Omron CX-Programmer project NuevoProyecto (CX-Programmer 9.61)

# PLC Caramelos: CJ2M CPU11

## Program NuevoPrograma1 (cyclic task 0)
Local symbols
CincoCent 1.01 BOOL  ; 1.01
DiezCent 1.02 BOOL  ; 1.02
Encender 0.00 BOOL  ; 0.00
ExpulsandoCaA 1.14 BOOL  ; 1.14
ExpulsandoCaB 1.15 BOOL  ; 1.15
IgualQueCinco 3.11 BOOL  ; 3.11
IgualQueDiez 3.12 BOOL  ; 3.12
IgualQueQuince 3.03 BOOL  ; 3.03
IgualQueVeinte 3.02 BOOL  ; 3.02
LedCarameloA 1.06 BOOL  ; 1.06
LedCarameloB 1.07 BOOL  ; 1.07
MasDeVeinte 1.05 BOOL  ; 1.05
MayorQueVeinte 3.10 BOOL  ; 3.10
MenorQueVeinte 3.01 BOOL  ; 3.01
P0 2.00 BOOL  ; 2.00
P1 2.01 BOOL  ; 2.01
P2 2.02 BOOL  ; 2.02
P3 2.03 BOOL  ; 2.03
P4 2.04 BOOL  ; 2.04
P5 2.05 BOOL  ; 2.05
P6 2.06 BOOL  ; 2.06
P7 2.07 BOOL  ; 2.07
P8 2.08 BOOL  ; 2.08
P9 2.09 BOOL  ; 2.09
Preparada 1.00 BOOL  ; 1.00
QuinceCent 1.03 BOOL  ; 1.03
Recuperar 0.11 BOOL  ; 0.11
Reset 2.10 BOOL  ; 2.10
SeleccionarCaA 0.14 BOOL  ; 0.14
SeleccionarCaB 0.15 BOOL  ; 0.15
SumaCinco 0.12 BOOL  ; 0.12
SumaDiez 0.13 BOOL  ; 0.13
VeinteCent 1.04 BOOL  ; 1.04

### Section Main

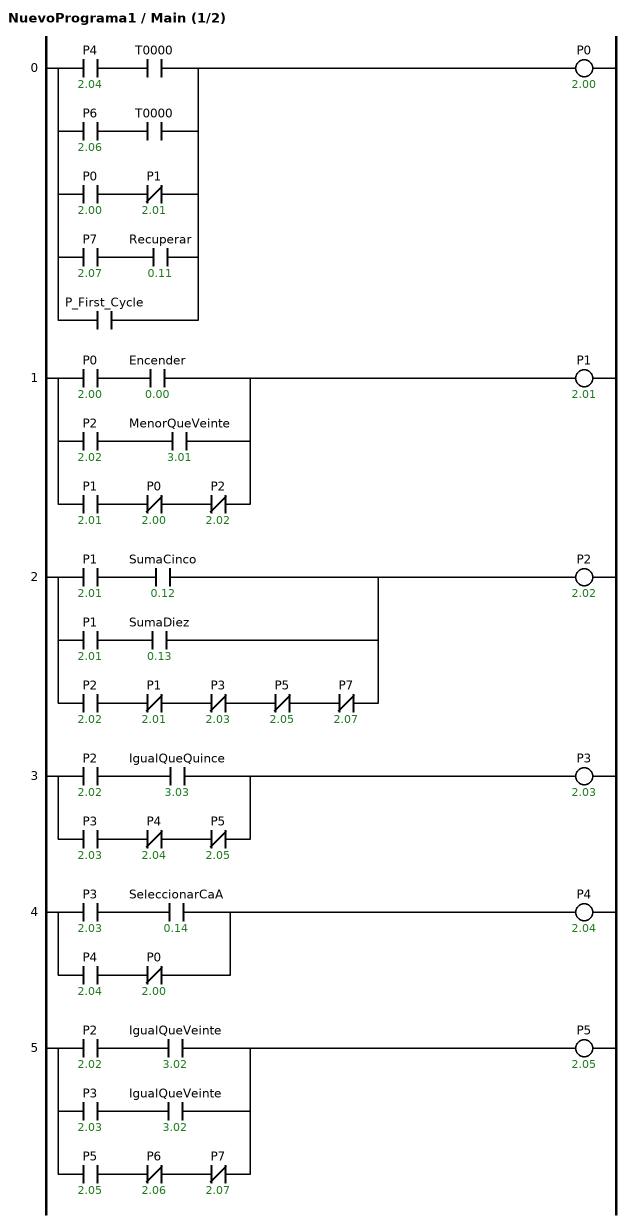
; rung 0
LD P4  ; 2.04
AND T0000
LD P6  ; 2.06
AND T0000
ORLD
LD P0  ; 2.00
ANDNOT P1  ; 2.01
ORLD
LD P7  ; 2.07
AND Recuperar  ; 0.11
ORLD
OR P_First_Cycle
OUT P0  ; 2.00
; rung 1
LD P0  ; 2.00
AND Encender  ; 0.00
LD P2  ; 2.02
AND MenorQueVeinte  ; 3.01
ORLD
LD P1  ; 2.01
ANDNOT P0  ; 2.00
ANDNOT P2  ; 2.02
ORLD
OUT P1  ; 2.01
; rung 2
LD P1  ; 2.01
AND SumaCinco  ; 0.12
LD P1  ; 2.01
AND SumaDiez  ; 0.13
ORLD
LD P2  ; 2.02
ANDNOT P1  ; 2.01
ANDNOT P3  ; 2.03
ANDNOT P5  ; 2.05
ANDNOT P7  ; 2.07
ORLD
OUT P2  ; 2.02
; rung 3
LD P2  ; 2.02
AND IgualQueQuince  ; 3.03
LD P3  ; 2.03
ANDNOT P4  ; 2.04
ANDNOT P5  ; 2.05
ORLD
OUT P3  ; 2.03
; rung 4
LD P3  ; 2.03
AND SeleccionarCaA  ; 0.14
LD P4  ; 2.04
ANDNOT P0  ; 2.00
ORLD
OUT P4  ; 2.04
; rung 5
LD P2  ; 2.02
AND IgualQueVeinte  ; 3.02
LD P3  ; 2.03
AND IgualQueVeinte  ; 3.02
ORLD
LD P5  ; 2.05
ANDNOT P6  ; 2.06
ANDNOT P7  ; 2.07
ORLD
OUT P5  ; 2.05

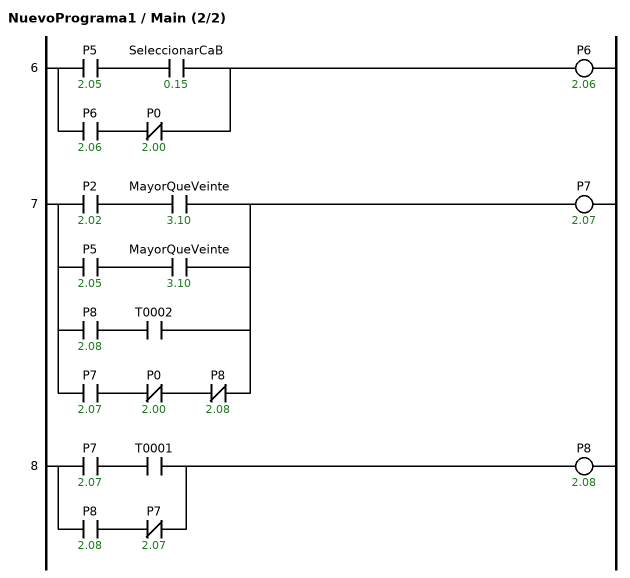
; rung 6
LD P5  ; 2.05
AND SeleccionarCaB  ; 0.15
LD P6  ; 2.06
ANDNOT P0  ; 2.00
ORLD
OUT P6  ; 2.06
; rung 7
LD P2  ; 2.02
AND MayorQueVeinte  ; 3.10
LD P5  ; 2.05
AND MayorQueVeinte  ; 3.10
ORLD
LD P8  ; 2.08
AND T0002
ORLD
LD P7  ; 2.07
ANDNOT P0  ; 2.00
ANDNOT P8  ; 2.08
ORLD
OUT P7  ; 2.07
; rung 8
LD P7  ; 2.07
AND T0001
LD P8  ; 2.08
ANDNOT P7  ; 2.07
ORLD
OUT P8  ; 2.08

### Section Comparadores

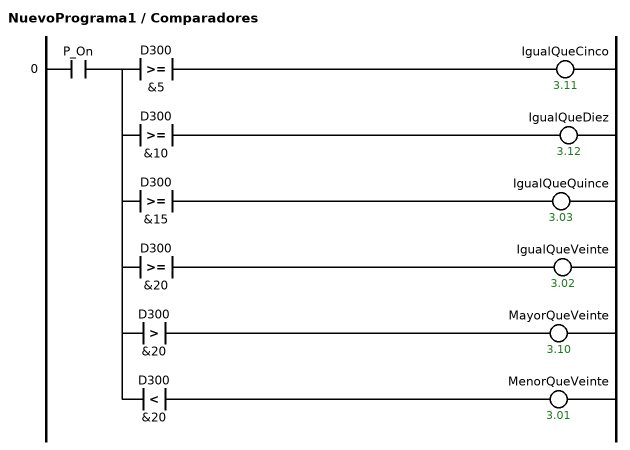
; rung 0
LD P_On
OUT TR0
AND>=(325) D300 &5
OUT IgualQueCinco  ; 3.11
LD TR0
AND>=(325) D300 &10
OUT IgualQueDiez  ; 3.12
LD TR0
AND>=(325) D300 &15
OUT IgualQueQuince  ; 3.03
LD TR0
AND>=(325) D300 &20
OUT IgualQueVeinte  ; 3.02
LD TR0
AND>(320) D300 &20
OUT MayorQueVeinte  ; 3.10
LD TR0
AND<(310) D300 &20
OUT MenorQueVeinte  ; 3.01

### Section Sumadores

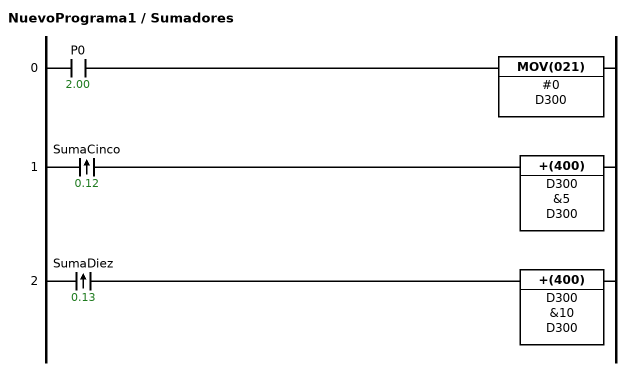
; rung 0
LD P0  ; 2.00
MOV(021) #0 D300
; rung 1
@LD SumaCinco  ; 0.12
+(400) D300 &5 D300
; rung 2
@LD SumaDiez  ; 0.13
+(400) D300 &10 D300

### Section Timers

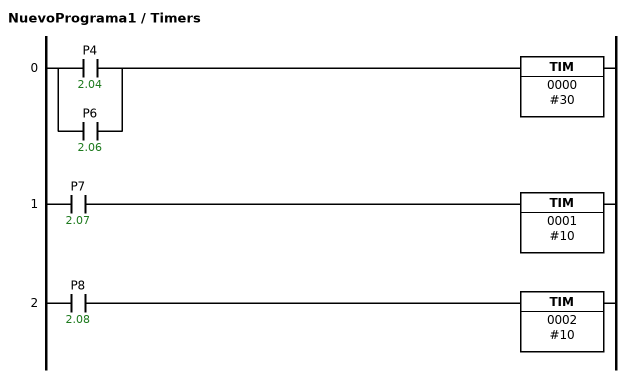
; rung 0
LD P4  ; 2.04
OR P6  ; 2.06
TIM 0000 #30
; rung 1
LD P7  ; 2.07
TIM 0001 #10
; rung 2
LD P8  ; 2.08
TIM 0002 #10

### Section Leds

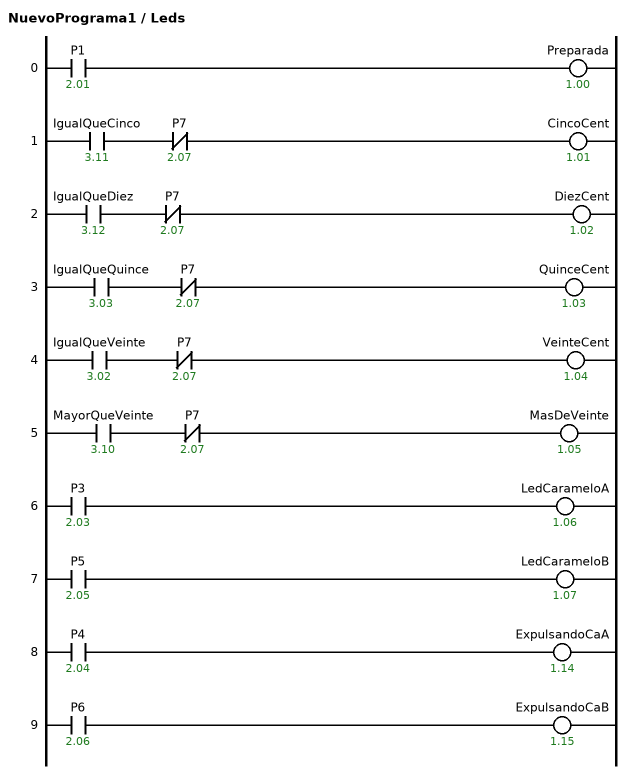
; rung 0
LD P1  ; 2.01
OUT Preparada  ; 1.00
; rung 1
LD IgualQueCinco  ; 3.11
ANDNOT P7  ; 2.07
OUT CincoCent  ; 1.01
; rung 2
LD IgualQueDiez  ; 3.12
ANDNOT P7  ; 2.07
OUT DiezCent  ; 1.02
; rung 3
LD IgualQueQuince  ; 3.03
ANDNOT P7  ; 2.07
OUT QuinceCent  ; 1.03
; rung 4
LD IgualQueVeinte  ; 3.02
ANDNOT P7  ; 2.07
OUT VeinteCent  ; 1.04
; rung 5
LD MayorQueVeinte  ; 3.10
ANDNOT P7  ; 2.07
OUT MasDeVeinte  ; 1.05
; rung 6
LD P3  ; 2.03
OUT LedCarameloA  ; 1.06
; rung 7
LD P5  ; 2.05
OUT LedCarameloB  ; 1.07
; rung 8
LD P4  ; 2.04
OUT ExpulsandoCaA  ; 1.14
; rung 9
LD P6  ; 2.06
OUT ExpulsandoCaB  ; 1.15

### Section END
; rung 0
END(001)